{attribute 'TcGenerated'}
{attribute 'no-analysis'}
{attribute 'linkalways'}
// This function has been automatically generated from the project information.
VAR_GLOBAL CONSTANT
	{attribute 'const_non_replaced'}
	stLibVersion_Tk_Diagnosis_EtherCAT : ST_LibVersion := (iMajor := 0, iMinor := 0, iBuild := 9, iRevision := 1, nFlags := 0, sVersion := '0.0.9.1');
END_VAR

(* stored: Version 1.1.0.1
   GVL Global_Version: Id {8f5b7fa3-b471-4ca6-9c6c-d3cb834e4751} *)
